TYPE ST_IOOutput :
STRUCT
	QxLampeRed AT%Q*:BOOL;
	QxLampeVerte AT%Q* : BOOL;
	QxLampeOrange AT%Q* :BOOL;
	
	
END_STRUCT
END_TYPE

(* stored: Version 1.1.0.1, ProductVersion 3.1.4020.12
   DUT ST_IOOutput: Id {d69b4ab8-e57a-466e-85fc-d2391d517834} *)
